FUNCTION_BLOCK ConveyorTracking
VAR_INPUT
	ProductPresent				:	BOOL;		// sensor detecting the product at the start of the conveyor
	ProductType					:	INT;		// product type
	EncoderResolution			:	REAL;		// how many mm distance per one encoder pulse [mm/pulses]
	Encoder						:	LINT;		// raw encoder value in pulses	
	TrackingAccuracy			:	REAL;		// needed product tracking accuracy [mm]
	DropPosition				:	UINT;		// diverter position in [mm]

	Reset						:	BOOL;		// reset all tracking logic
END_VAR
VAR_OUTPUT
	DiverterCmd					:	BOOL;		// command to activate the diverter
	DistanceMoved				:	REAL;		// distance a product has moved since product presence sensor
END_VAR
VAR
	Init						:	BOOL:=TRUE;
	EncValueMem					:	LINT;
	EncDiff						: 	LINT;
	
	rtTrack						: 	R_TRIG;
	TrackTrigger				: 	BOOL;
	
	Register					:	ARRAY[0..500] OF stShiftRegData;
	ShiftRegister01				: 	ShiftRegister;
	ctuProductLen				: 	CTU;
	ftrigProduct				: 	F_TRIG;
	ProductLen					:	WORD;
	FifoLoad					: 	Fifo;
	MiddlePointPos				: 	REAL;

	rtrigProductPresent			: 	R_TRIG;
	ProductStarted				: 	BOOL;
	ftrigProductGone			: 	F_TRIG;
END_VAR
VAR // added by the converter: edge detectors and wires of the graphical bodies
    _w1, _w2 : BOOL;
END_VAR

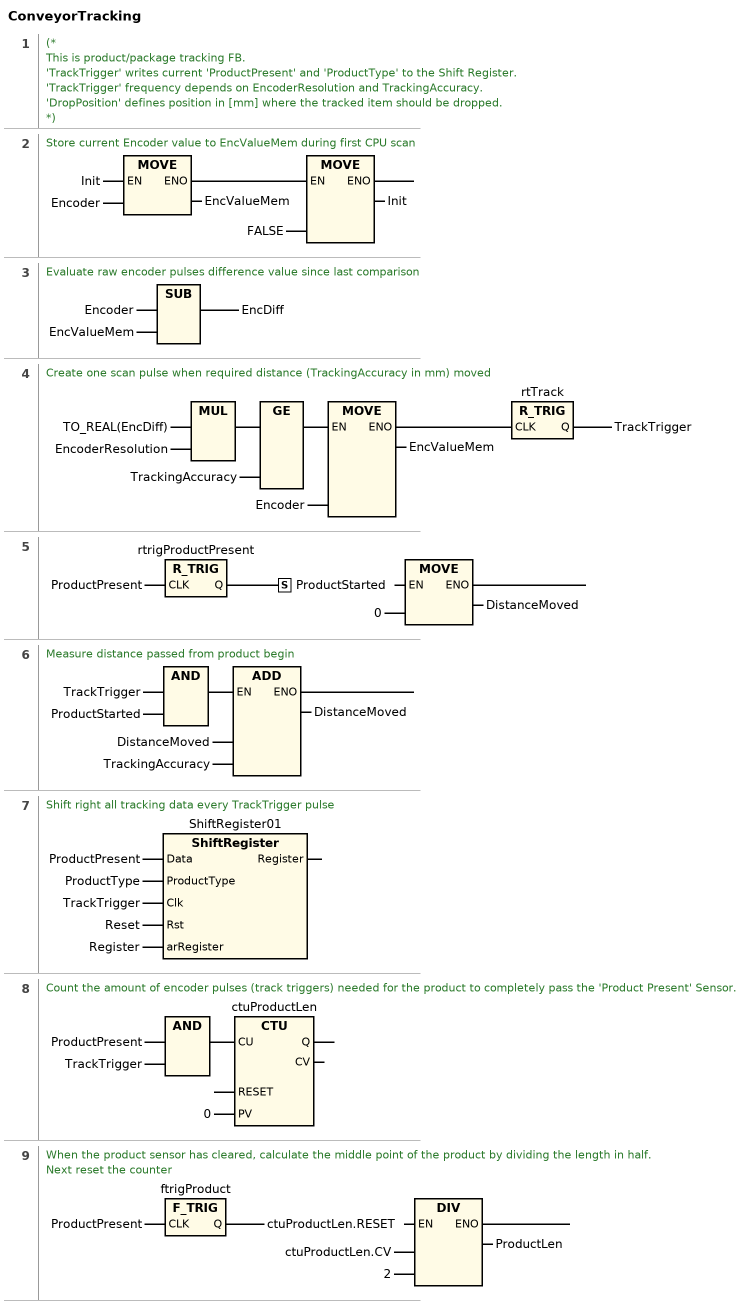
// NETWORK 1
// (*
// This is product/package tracking FB.
// 'TrackTrigger' writes current 'ProductPresent' and 'ProductType' to the Shift Register.
// 'TrackTrigger' frequency depends on EncoderResolution and TrackingAccuracy.
// 'DropPosition' defines position in [mm] where the tracked item should be dropped.
// *)

// NETWORK 2
// Store current Encoder value to EncValueMem during first CPU scan
_w1 := Init;
IF _w1 THEN EncValueMem := Encoder; END_IF
IF _w1 THEN Init := FALSE; END_IF

// NETWORK 3
// Evaluate raw encoder pulses difference value since last comparison
EncDiff := Encoder - EncValueMem;

// NETWORK 4
// Create one scan pulse when required distance (TrackingAccuracy in mm) moved
_w2 := (TO_REAL(EncDiff)) * EncoderResolution >= TrackingAccuracy;
IF _w2 THEN EncValueMem := Encoder; END_IF
rtTrack(CLK := _w2); // R_TRIG
TrackTrigger := rtTrack.Q;

// NETWORK 5
rtrigProductPresent(CLK := ProductPresent); // R_TRIG
ProductStarted S= rtrigProductPresent.Q;
IF rtrigProductPresent.Q THEN DistanceMoved := 0; END_IF

// NETWORK 6
// Measure distance passed from product begin
IF TrackTrigger AND ProductStarted THEN DistanceMoved := DistanceMoved + TrackingAccuracy; END_IF

// NETWORK 7
// Shift right all tracking data every TrackTrigger pulse
ShiftRegister01(
    Data := ProductPresent,
    ProductType := ProductType,
    Clk := TrackTrigger,
    Rst := Reset,
    arRegister := Register); // ShiftRegister

// NETWORK 8
// Count the amount of encoder pulses (track triggers) needed for the product to completely pass the 'Product Present' Sensor.
ctuProductLen(CU := ProductPresent AND TrackTrigger, PV := 0); // CTU

// NETWORK 9
// When the product sensor has cleared, calculate the middle point of the product by dividing the length in half.
// Next reset the counter
ftrigProduct(CLK := ProductPresent); // F_TRIG
ctuProductLen.RESET := ftrigProduct.Q;
IF ftrigProduct.Q THEN ProductLen := ctuProductLen.CV / 2; END_IF

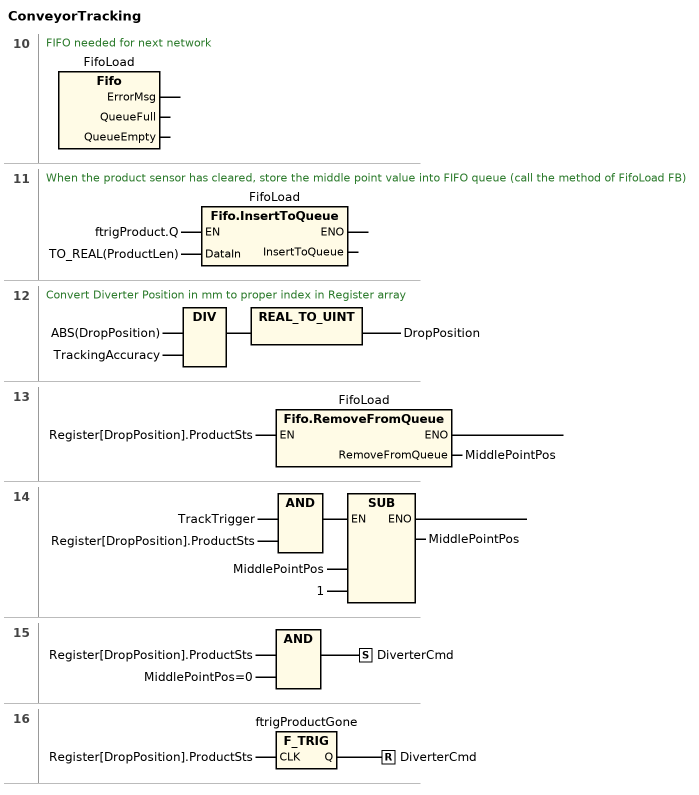
// NETWORK 10
// FIFO needed for next network
FifoLoad(); // Fifo

// NETWORK 11
// When the product sensor has cleared, store the middle point value into FIFO queue (call the method of FifoLoad FB)
IF ftrigProduct.Q THEN FifoLoad.InsertToQueue(DataIn := TO_REAL(ProductLen)); END_IF

// NETWORK 12
// Convert Diverter Position in mm to proper index in Register array
DropPosition := REAL_TO_UINT((ABS(DropPosition)) / TrackingAccuracy);

// NETWORK 13
IF Register[DropPosition].ProductSts THEN FifoLoad.RemoveFromQueue(RemoveFromQueue => MiddlePointPos); END_IF

// NETWORK 14
IF TrackTrigger AND Register[DropPosition].ProductSts THEN MiddlePointPos := MiddlePointPos - 1; END_IF

// NETWORK 15
DiverterCmd S= Register[DropPosition].ProductSts AND (MiddlePointPos=0);

// NETWORK 16
ftrigProductGone(CLK := Register[DropPosition].ProductSts); // F_TRIG
DiverterCmd R= ftrigProductGone.Q;

END_FUNCTION_BLOCK

(* stored: Version 1.1.0.1, ProductVersion 3.1.4024.15
   POU ConveyorTracking: Id {27cd897f-92c3-4014-8095-c4c10f172c4d}, SpecialFunc None *)
